# EPICS autosave request: iocBoot/gmca_23b_ioc1/dbSave/robot.req
% $(P)pause
$(P)gh_pos
$(P)gy_pos
$(P)tmoh
$(P)tmow
$(P)tmoc
$(P)senh
$(P)senb
$(P)senc
$(P)send
$(P)warmup_duration
